(* IEC 61131-3 sources: programs/VI-54/VI-54_20171205/VI-54_20171205/Stations/PLC_VI54/VI-54_171014/Class/_DriveActValues, 1 file *)

(* ---- _DriveActValues.st ---- *)
(*!
<Class
	Name               = "_DriveActValues"
	Revision           = "1.13"
	RealtimeTask       = "false"
	CyclicTask         = "true"
	DefCyclictime      = "100 ms"
	BackgroundTask     = "false"
	Sigmatek           = "true"
	OSInterface        = "false"
	HighPriority       = "false"
	Automatic          = "false"
	UpdateMode         = "Prescan"
	IconPath           = ".\Class\_DriveMngBase\Drive.ico"
	SharedCommandTable = "true"
	Objectsize         = "(570,1920)"
	Comment            = "displays the actual values of the connected Drive">
	<Channels>
		<Server Name="I_BCC" Visualized="true" Initialize="false" WriteProtected="true" Retentive="false" Comment="Para-Nr : 182&#13;&#10;Unit  : [-]&#13;&#10;Checksum of all parameters for data integrity check&#13;&#10;"/>
		<Server Name="I_BITS" Visualized="true" Initialize="false" WriteProtected="true" Retentive="false" Comment="Para-Nr : 205&#13;&#10;Unit  : [-]&#13;&#10;BIT 0 ... PLL BIT0:&#13;&#10;BIT 1 ... PLL BIT1:&#13;&#10;00=PLL locked;&#13;&#10;01=PLL locked, more than half of the pll range is used (frequency to high);&#13;&#10;10=PLL locked, less than half of the pll range is used (frequency to low);&#13;&#10;11=PLL not locked&#13;&#10;BIT 2 ... Digital Input 6: LOCK &amp; ENABLE &amp; ENABLE_BRAKE&#13;&#10;BIT 3 ... IGBT Voltage (LOCK)&#13;&#10;BIT 4 ... ENABLE Input&#13;&#10;BIT 5 ... ENABLE_BRAKE Input&#13;&#10;BIT 6 ... Digital Input 1&#13;&#10;BIT 7 ... Digital Input 2&#13;&#10;BIT 8 ... Digital Input 3&#13;&#10;BIT 9 ... Digital Input 4&#13;&#10;BIT10 ... Digital Input 5"/>
		<Server Name="I_CAP" Visualized="true" Initialize="false" WriteProtected="true" Retentive="false" Comment="Para-Nr : 202&#13;&#10;Unit  : [-]&#13;&#10;Motorposition at the last edge of the capture input&#13;&#10;The selection of the input and the edge (rising/falling) is done by [A-CAPREF].&#13;&#10;&#13;&#10;If a capture happens, the corresponding bit in the statusword is toggled (statusword see [A-VALTT1] and [A-VALTT2]).&#13;&#10;"/>
		<Server Name="I_CAP4" Visualized="true" Initialize="false" WriteProtected="true" Retentive="false" Comment="Para-Nr : 203&#13;&#10;Unit  : [-]&#13;&#10;Motorposition at the last edge of the common capture input 4&#13;&#10;&#13;&#10;If a capture happens, the corresponding bit in the statusword is toggled (statusword see [A-VALTT1] and [A-VALTT2])."/>
		<Server Name="I_CAPENC" Visualized="true" Initialize="false" WriteProtected="true" Retentive="false" Comment="Para-Nr : 204&#13;&#10;Unit  : [-]&#13;&#10;Position of the second encoder at the last edge at the capture input&#13;&#10;The selection of the input and the edge (rising/falling) is done by A-CAPREF.&#13;&#10;&#13;&#10;If a capture happens, the corresponding bit in the statusword is toggled (statusword see A-VALTT1 and A-VALTT2)."/>
		<Server Name="I_DERROR" Visualized="true" Initialize="false" WriteProtected="true" Retentive="false" Comment="Para-Nr : 201&#13;&#10;Unit  : [-]&#13;&#10;Description : Internal Drive Errors&#13;&#13;&#10;&#13;&#13;&#10;MDD,SDD - Drives &#13;&#10;=============================================================================================&#13;&#10;Bit   0 SSI_ERROR (not supported by MDD 100)(additional Information to the Host Communication Error in [I-STATUS])&#13;&#10;Bit   1 HOST_ERROR (not supported by MDD 100)(additional Information to the Host Communication Error in [I-STATUS])&#13;&#10;Bit   2 SHORT_ERROR (short of the power stage)&#13;&#10;Bit   3 RAM_ERROR (error in the code ram area)&#13;&#10;Bit   4 FPGA_WATCHDOG_ERROR (not supported by MDD 100)(is set by the fpga watchdog mechanism)&#13;&#10;Bit   5 ADOFF_ERROR (not supported by MDD 100)(the offset of the motor current is to high)&#13;&#10;Bit   6 VCC18_ERROR (Phasing Direction Error, set when the motor turns in the wrong direction after commutation)&#13;&#10;Bit   7 VCCE_ERROR (Internal Encoder Error)&#13;&#10;Bit   8 ASMFU_IMAX_ERROR (is set if the asynchronous motor current is to high)&#13;&#10;Bit   9 PHASING_SIGNAL_STRENGTH_ERROR (Phasing Signal Strengh Error, more detailed information in Drive help parameter description I-DERROR)&#13;&#10;Bit  10 PHASING_POSITION_ERROR (is set when the position of the motor changes too drastically durin commutation)&#13;&#10;Bit  11 REGEN_ERROR (is set if the regen resistor can not be turned off)&#13;&#10;Bit  12 ENCODER_COUNTER_ERROR (not supported by MDD 100)(is set if the encoder counter check detects a fault)&#13;&#10;Bit  13 SIN_COS_COMMUT_ERROR (is set if a communication error exceeds 50ms)&#13;&#10;Bit  14 LVDS_ERROR (MDD only, is set if a communication error occurs between master and slave)&#13;&#10;Bit  15 PHASING_PHASE_SHIFT_ERROR (is set when the distance between the maximum positive/negative feedback peaks does not equal 180° +- 8°)&#13;&#10;Bit  16 PHASING_FOURIER_SIGNAL_ERROR (fourier signal cannot be calculated)&#13;&#10;&#13;&#10;DC06x&#13;&#10;=============================================================================================&#13;&#10;Bit   2 SHORT_ERROR (short of the power stage)&#13;&#10;Bit  13 FEEDBACK_ADC (feedback resolver values are not valid)(only DC061)&#13;&#10;Bit  15 SAFETY_ERROR  (safety error)&#13;&#10;Bit  16 SAFETY_WARNING (safety warning) &#13;&#10;Bit  21 Z_IMPULS_ERROR  (the z-impuls did not appeared within the time frame) (only DC062)&#13;&#10;Bit  23 FEEDBACK_SUPPLY (the feedback supply voltage fell below 15V)(only DC062)&#13;&#10;&#13;&#10;&#13;&#10;For more detailed informations, look at the parameter description of I-DERROR (201) in the Drive Help.&#13;&#13;&#10;These bits cause the Drive Error Ramp/Drive Error No Ramp in [I-STATUS]."/>
		<Server Name="I_FBB" Visualized="true" Initialize="false" WriteProtected="true" Retentive="false" Comment="Para-Nr : 208&#13;&#10;Unit  : [-]&#13;&#10;Actual value Feedback bits&#13;&#10;&#13;&#10;Bit0: Toggle status bit for the cyclic monitoring of the error status for EnDat and Hiperface encoders. See A-FB.&#13;&#10;Bit1: Status bit for the K-FBRW 5 command (Read offset from encoder). If this command was executed, Bit1 = 1. &#13;&#10;Bit2..15: Reserve&#13;&#10;Bit16..31: In these 2 bytes, the internal encoder error codes are stored as long as the K-FBRW 4 command was executed or the cyclic error status monitor is active (A-FB).&#13;&#10;"/>
		<Server Name="I_FPOS" Visualized="true" Initialize="false" WriteProtected="true" Retentive="false" Comment="Para-Nr : 177&#13;&#10;Unit  : [-]&#13;&#10;Description : Resolver angle&#13;&#10;&#13;&#10;"/>
		<Server Name="I_I2T" Visualized="true" Initialize="false" WriteProtected="true" Retentive="false" Comment="Para-Nr : 193&#13;&#10;Unit  : [%]&#13;&#10;Description : Actual value of I2T of the power stage in % of [C-ICONT]&#13;&#13;&#10;&#13;&#13;&#10;The i2t-mechanism of the drive limits the current and the continuous current is always limited to the value of [C-ICONT].&#13;&#10;"/>
		<Server Name="I_IA" Visualized="true" Initialize="false" WriteProtected="true" Retentive="false" Comment="Para-Nr : 178 &#13;&#10;Unit  : [-]&#13;&#10;AD-value Ia (only for test purpose)&#13;&#10;"/>
		<Server Name="I_IB" Visualized="true" Initialize="false" WriteProtected="true" Retentive="false" Comment="Para-Nr : 179&#13;&#10;Unit  : [-]&#13;&#10;AD-value Ib (only for test purpose)"/>
		<Server Name="I_ICMD" Visualized="true" Initialize="false" WriteProtected="true" Retentive="false" Comment="Para-Nr : 194&#13;&#10;Unit  : [mA]&#13;&#10;Description : Current set point in Q - direction"/>
		<Server Name="I_ICONT" Visualized="true" Initialize="false" WriteProtected="true" Retentive="false" Comment="Para-Nr : 186&#13;&#10;Unit  : [mA]&#13;&#10;Description : Drive continuos current&#13;&#10;"/>
		<Server Name="I_ID" Visualized="true" Initialize="false" WriteProtected="true" Retentive="false" Comment="Para-Nr : 192&#13;&#10;Unit  : [mA]&#13;&#10;Description : Actual value of the current in D - direction&#13;&#10;"/>
		<Server Name="I_INT1" Visualized="true" Initialize="false" WriteProtected="true" Retentive="false" Comment="Para-Nr : 206&#13;&#10;Unit  : [-]&#13;&#10;Internal Actual Value 1&#13;&#10;&#13;&#10;A-INT1 defines which internal actual value is displayed here.&#13;&#10;&#13;&#10;See also I-INT2."/>
		<Server Name="I_INT2" Visualized="true" Initialize="false" WriteProtected="true" Retentive="false" Comment="Para-Nr : 207&#13;&#10;Unit  : [-]&#13;&#10;Internal Actual Value 2&#13;&#10;&#13;&#10;A-INT2 defines which internal actual value is displayed here.&#13;&#10;&#13;&#10;See also I-INT1."/>
		<Server Name="I_IPEAK" Visualized="true" Initialize="false" WriteProtected="true" Retentive="false" Comment="Para-Nr : 185&#13;&#10;Unit  : [mA]&#13;&#10;Description : Drive peak current&#13;&#10;"/>
		<Server Name="I_IQ" Visualized="true" Initialize="false" WriteProtected="true" Retentive="false" Comment="Para-Nr : 191&#13;&#10;Unit  : [mA]&#13;&#10;Description : Actual value of the current in Q - direction&#13;&#10;"/>
		<Server Name="I_MPOS" Visualized="true" Initialize="false" WriteProtected="true" Retentive="false" Comment="Para-Nr : 180&#13;&#10;Unit  : [-]&#13;&#10;Description : Actual multiturn position  in 1/8 of a revolution (available only with [M-TYPE] = 1)"/>
		<Server Name="I_N" Visualized="true" Initialize="false" WriteProtected="true" Retentive="false" Comment="Para-Nr : 197&#13;&#10;Unit  : [rpm]&#13;&#10;Description : Actual speed unsmoothed&#13;&#10;"/>
		<Server Name="I_NCMD" Visualized="true" Initialize="false" WriteProtected="true" Retentive="false" Comment="Para-Nr : 190&#13;&#10;Unit  : [rpm]&#13;&#10;Description : Speed set point&#13;&#10;"/>
		<Server Name="I_NFILT" Visualized="true" Initialize="false" WriteProtected="true" Retentive="false" Comment="Para-Nr : 198&#13;&#10;Unit  : [rpm]&#13;&#10;Description : Actual speed smoothed by [V-T]&#13;&#10;"/>
		<Server Name="I_PBAL" Visualized="true" Initialize="false" WriteProtected="true" Retentive="false" Comment="Para-Nr : 196&#13;&#10;Unit  : [W]&#13;&#10;Description : Actual regen power&#13;&#13;&#10;This value is influenced by [G-RBAL].&#13;&#10;"/>
		<Server Name="I_PCMD" Visualized="true" Initialize="false" WriteProtected="true" Retentive="false" Comment="Para-Nr : 174&#13;&#10;Unit  : [-]&#13;&#10;Description : Position setpoint&#13;&#10;"/>
		<Server Name="I_PE" Visualized="true" Initialize="false" WriteProtected="true" Retentive="false" Comment="Para-Nr : 175&#13;&#10;Unit  : [-]&#13;&#10;Description : Position error&#13;&#10;&#13;&#10;"/>
		<Server Name="I_POS" Visualized="true" Initialize="false" WriteProtected="true" Retentive="false" Comment="Para-Nr : 176&#13;&#10;Unit  : [-]&#13;&#10;Description : Actual position (internal 64 bit position scaled by [P-PSCALE])&#13;&#10;&#13;&#10;"/>
		<Server Name="I_STATUS" Visualized="true" Initialize="false" WriteProtected="true" Retentive="false" Comment="Para-Nr : 199&#13;&#10;Unit  : [-]&#13;&#10;Description : Status register:&#13;&#13;&#10;&#13;&#13;&#10;Bit  0   Mains phase (1-phase supply)&#13;&#10;Bit  1   Mains fault&#13;&#10;Bit  2   Motor axis over-current&#13;&#10;Bit  3   Over voltage DC-Link&#13;&#10;Bit  4   Under voltage DC-link&#13;&#10;Bit  5   Motor axis phase failure&#13;&#10;Bit  6   Holding brake error&#13;&#10;Bit  7   Holding brake switch damaged&#13;&#10;Bit  8   reserved&#13;&#10;Bit  9   Motor thermostat&#13;&#10;Bit 10  Ambient temperature&#13;&#10;Bit 11  Heat sink temperature&#13;&#10;Bit 12  Feedback Error&#13;&#10;Bit 13  Commutation error&#13;&#10;Bit 14  Over speed&#13;&#10;Bit 15  Contouring Error&#13;&#10;Bit 16  Trajectory Error&#13;&#10;Bit 17  Host Communication Error&#13;&#10;Bit 18  Drive Error Ramp, for additional information see [I-DERROR]&#13;&#10;Bit 19  Drive Error No Ramp, for additional information see [I-DERROR]&#13;&#10;Bit 20  External Enable Locked Error&#13;&#10;Bit 21  IGBT Driver Voltage Error&#13;&#10;Bit 22  max. Regen Power Error&#13;&#10;Bit 23  24V Brake Supply Error&#13;&#10;Bit 24  reserved&#13;&#10;Bit 25  I2T-Error&#13;&#10;Bit 26  Motor Temperature Warning&#13;&#10;Bit 27  Motor Parameter Error&#13;&#10;Bit 28  Multi-Turn Position Error&#13;&#10;Bit 29  Max Sum Power Limitation&#13;&#10;Bit 30  Speed Controler in Saturation&#13;&#10;Bit 31  Fan Error &#13;&#10;&#13;&#13;&#10;The masks  [G-MASKE1], [G-MASKE2], [G-MASKW] and [G-MASKD] &#13;&#10;define if the corresponding bit of I-STATUS causes a cast of the motor, a ramp stop of the motor, a warning or nothing.&#13;&#13;&#10;This errors can be cleared with [K-CLRF].&#13;&#10;For more detailed informations, look at the parameter description of I-STATUS(199) in the Drive Help.&#13;&#10;"/>
		<Server Name="I_TEMPE" Visualized="true" Initialize="false" WriteProtected="true" Retentive="false" Comment="Para-Nr : 184&#13;&#10;Unit  : [°C]&#13;&#10;Description : Actual ambient temperature&#13;&#10;"/>
		<Server Name="I_TEMPK" Visualized="true" Initialize="false" WriteProtected="true" Retentive="false" Comment="Para-Nr : 183&#13;&#10;Unit  : [°C]&#13;&#10;Description : Actual heat sink temperature&#13;&#10;&#13;&#10;"/>
		<Server Name="I_TEMPM" Visualized="true" Initialize="false" WriteProtected="true" Retentive="false" Comment="Para-Nr : 181&#13;&#10;Unit  : [Ohm]&#13;&#10;Description : Actual value of the PTC in the motor winding &#13;&#10;"/>
		<Server Name="I_VBUS" Visualized="true" Initialize="false" WriteProtected="true" Retentive="false" Comment="Para-Nr : 195&#13;&#10;Unit  : [V]&#13;&#10;Description : Actual DC-link voltage&#13;&#10;"/>
	</Channels>
	<RevDoku>
		<Owner Company="Sigmatek" Author="HasHan"/>
		<Dokumentation Revision="1.13" Date="08.11.2016" Author="ZoePat" Company="Sigmatek" Description="Client &quot;DriveAxis&quot; is now not required."/>
		<Dokumentation Revision="1.12" Date="16.06.2015" Author="EisMic" Company="Sigmatek" Description="Updated description from I-STATUSand I-DERROR Bits."/>
		<Dokumentation Revision="1.11" Date="06.10.2014" Author="LanSte" Company="Sigmatek" Description="Added support for drive parameters P208 amd P122"/>
		<Dokumentation Revision="1.10" Date="04.12.2013" Author="ObeChr" Company="Sigmatek" Description="Added missing Bits in Type for Server I-STATUS + I-DERROR"/>
		<Dokumentation Revision="1.0" Date="05.08.2009" Author="HasHan" Company="Sigmatek" Description="Creation"/>
	</RevDoku>
	<Network Name="_DriveActValues">
		<!-- List of Components in this network -->
		<Components>
			<Object
				Name       = "_base"
				Class      = "_DriveParaBase"
				Position   = "(218,120)"
				Visualized = "false">
				<Channels>
					<Server Name="State"/>
					<Client Name="DriveAxis"/>
					<Client Name="ErrorCode"/>
				</Channels>
			</Object>
		</Components>
		<Comments>
		</Comments>
		<!-- List of Connections in this network -->
		<Connections>
			<Connection Source="this.State" Destination="_base.State" Vertices="(740,210),(568,210),"/>
			<Connection Source="_base.DriveAxis" Destination="this.DriveAxis" Vertices="(218,210),(38,210),"/>
			<Connection Source="_base.ErrorCode" Destination="this.ErrorCode" Vertices="(218,270),(38,270),"/>
		</Connections>
		<!-- Headerfiles -->
		<Options>
		</Options>
	</Network>
</Class>
*)
#pragma using _DriveParaBase

_DriveActValues : CLASS
: _DriveParaBase
  //Servers:
	I_PCMD 	: SvrCh_DINT;
	I_PE 	: SvrCh_DINT;
	I_POS 	: SvrCh_DINT;
	I_FPOS 	: SvrCh_DINT;
	I_MPOS 	: SvrCh_DINT;
	I_TEMPM 	: SvrCh_DINT;
	I_TEMPK 	: SvrCh_DINT;
	I_TEMPE 	: SvrCh_DINT;
	I_IPEAK 	: SvrCh_DINT;
	I_ICONT 	: SvrCh_DINT;
	I_NCMD 	: SvrCh_DINT;
	I_IQ 	: SvrCh_DINT;
	I_ID 	: SvrCh_DINT;
	I_I2T 	: SvrCh_DINT;
	I_ICMD 	: SvrCh_DINT;
	I_VBUS 	: SvrCh_DINT;
	I_PBAL 	: SvrCh_DINT;
	I_N 	: SvrCh_DINT;
	I_NFILT 	: SvrCh_DINT;
	I_STATUS 	: SvrCh__SDDISTATE;
	I_DERROR 	: SvrCh__SDDIDERROR;
	I_BCC 	: SvrCh_DINT;
	I_IA 	: SvrCh_DINT;
	I_IB 	: SvrCh_DINT;
	I_CAP 	: SvrCh_DINT;
	I_CAP4 	: SvrCh_DINT;
	I_CAPENC 	: SvrCh_DINT;
	I_BITS 	: SvrCh_DINT;
	I_INT1 	: SvrCh_DINT;
	I_INT2 	: SvrCh_DINT;
	I_FBB 	: SvrCh_DINT;
  //Clients:
  //Variables:
		TimeMarkFast 	: UDINT;
		ActValSSW 	: DINT;
		bdActValActive : BDINT
		[
		  1 bI_PCMD,
		  2 bI_PE,
		  3 bI_POS,
		  4 bI_FPOS,
		  5 bI_MPOS,
		  6 bI_TEMPM,
		  7 bI_TEMPK,
		  8 bI_TEMPE,
		  9 bI_IPEAK,
		  10 bI_ICONT,
		  11 bI_NCMD,
		  12 bI_IQ,
		  13 bI_ID,
		  14 bI_I2T,
		  15 bI_ICMD,
		  16 bI_VBUS,
		  17 bI_PBAL,
		  18 bI_N,
		  19 bI_NFILT,
		  20 I_STATUS,
		  21 bI_I_DERROR,
		];

  //Functions:

	FUNCTION VIRTUAL GLOBAL Init;

	FUNCTION VIRTUAL GLOBAL CyWork
		VAR_INPUT
			EAX 	: UDINT;
		END_VAR
		VAR_OUTPUT
			state (EAX) 	: UDINT;
		END_VAR;

	FUNCTION VIRTUAL GLOBAL RefreshPara
		VAR_INPUT
			usParaNr 	: USINT;
			dValue 	: DINT;
		END_VAR;

	FUNCTION GLOBAL ActValProc;
  //Tables:
	FUNCTION @STD
		VAR_OUTPUT
			ret_code	: CONFSTATES;
		END_VAR;
	FUNCTION GLOBAL TAB @CT_;
END_CLASS;

FUNCTION VIRTUAL GLOBAL _DriveActValues::CyWork
	VAR_INPUT
		EAX 	: UDINT;
	END_VAR
	VAR_OUTPUT
		state (EAX) 	: UDINT;
	END_VAR

	state:= READY;

  if (IsAxisConnected() = TRUE) & (DriveAxis.AxOkay() = true) & (DriveAxis.IsOnline() = true) then
    ActValProc();
    if DriveAxis <> READY then
      DriveAxis := READY;
    end_if;
  else
    this^.State  := ERROR;
    DriveAxis    := ERROR;
    ActValSSW    := SDD_I_PCMD;
    AnzASyncPara := 0;
  end_if;

END_FUNCTION

FUNCTION GLOBAL _DriveActValues::ActValProc

  if ops.tabsolute - TimeMarkFast >= ACTVALTIMEFAST then

    TimeMarkFast := ops.tabsolute;
    case ActValSSW of
    SDD_I_PCMD :
      SetASyncCmd(ParaNr:= SDD_I_PCMD, ParaRdWr:= 0, ParaValue:= 0, pThis:= this);
      ActValSSW := SDD_I_PE;

    SDD_I_PE :
      SetASyncCmd(ParaNr:= SDD_I_PE, ParaRdWr:= 0, ParaValue:= 0, pThis:= this);
      ActValSSW := SDD_I_POS;

    SDD_I_POS :
      SetASyncCmd(ParaNr:= SDD_I_POS, ParaRdWr:= 0, ParaValue:= 0, pThis:= this);
      ActValSSW := SDD_I_FPOS;

    SDD_I_FPOS :
      SetASyncCmd(ParaNr:= SDD_I_FPOS, ParaRdWr:= 0, ParaValue:= 0, pThis:= this);
      ActValSSW := SDD_I_MPOS;

    SDD_I_MPOS :
      SetASyncCmd(ParaNr:= SDD_I_MPOS, ParaRdWr:= 0, ParaValue:= 0, pThis:= this);
      ActValSSW := SDD_I_TEMPM;

    SDD_I_TEMPM :
      SetASyncCmd(ParaNr:= SDD_I_TEMPM, ParaRdWr:= 0, ParaValue:= 0, pThis:= this);
      ActValSSW := SDD_I_TEMPK;

    SDD_I_TEMPK :
      SetASyncCmd(ParaNr:= SDD_I_TEMPK, ParaRdWr:= 0, ParaValue:= 0, pThis:= this);
      ActValSSW := SDD_I_TEMPE;

    SDD_I_TEMPE :
      SetASyncCmd(ParaNr:= SDD_I_TEMPE, ParaRdWr:= 0, ParaValue:= 0, pThis:= this);
      ActValSSW := SDD_I_IPEAK;

    SDD_I_IPEAK :
      SetASyncCmd(ParaNr:= SDD_I_IPEAK, ParaRdWr:= 0, ParaValue:= 0, pThis:= this);
      ActValSSW := SDD_I_ICONT;

    SDD_I_ICONT :
      SetASyncCmd(ParaNr:= SDD_I_ICONT, ParaRdWr:= 0, ParaValue:= 0, pThis:= this);
      ActValSSW := SDD_I_NCMD;

    SDD_I_NCMD :
      SetASyncCmd(ParaNr:= SDD_I_NCMD, ParaRdWr:= 0, ParaValue:= 0, pThis:= this);
      ActValSSW := SDD_I_IQ;

    SDD_I_IQ :
      SetASyncCmd(ParaNr:= SDD_I_IQ, ParaRdWr:= 0, ParaValue:= 0, pThis:= this);
      ActValSSW := SDD_I_ID;

    SDD_I_ID :
      SetASyncCmd(ParaNr:= SDD_I_ID, ParaRdWr:= 0, ParaValue:= 0, pThis:= this);
      ActValSSW := SDD_I_I2T;

    SDD_I_I2T :
      SetASyncCmd(ParaNr:= SDD_I_I2T, ParaRdWr:= 0, ParaValue:= 0, pThis:= this);
      ActValSSW := SDD_I_ICMD;

    SDD_I_ICMD :
      SetASyncCmd(ParaNr:= SDD_I_ICMD, ParaRdWr:= 0, ParaValue:= 0, pThis:= this);
      ActValSSW := SDD_I_VBUS;

    SDD_I_VBUS :
      SetASyncCmd(ParaNr:= SDD_I_VBUS, ParaRdWr:= 0, ParaValue:= 0, pThis:= this);
      ActValSSW := SDD_I_PBAL;

    SDD_I_PBAL :
      SetASyncCmd(ParaNr:= SDD_I_PBAL, ParaRdWr:= 0, ParaValue:= 0, pThis:= this);
      ActValSSW := SDD_I_N;

    SDD_I_N :
      SetASyncCmd(ParaNr:= SDD_I_N, ParaRdWr:= 0, ParaValue:= 0, pThis:= this);
      ActValSSW := SDD_I_NFILT;

    SDD_I_NFILT :
      SetASyncCmd(ParaNr:= SDD_I_NFILT, ParaRdWr:= 0, ParaValue:= 0, pThis:= this);
      ActValSSW := SDD_I_STATUS;

    SDD_I_STATUS :
      SetASyncCmd(ParaNr:= SDD_I_STATUS, ParaRdWr:= 0, ParaValue:= 0, pThis:= this);
      ActValSSW := SDD_I_DERROR;

    SDD_I_DERROR :
      SetASyncCmd(ParaNr:= SDD_I_DERROR, ParaRdWr:= 0, ParaValue:= 0, pThis:= this);
      ActValSSW := SDD_I_CAP;

    SDD_I_CAP :
      SetASyncCmd(ParaNr:= SDD_I_CAP, ParaRdWr:= 0, ParaValue:= 0, pThis:= this);
      ActValSSW := SDD_I_CAP4;

    SDD_I_CAP4 :
      SetASyncCmd(ParaNr:= SDD_I_CAP4, ParaRdWr:= 0, ParaValue:= 0, pThis:= this);
      ActValSSW := SDD_I_CAPENC;

    SDD_I_CAPENC :
      SetASyncCmd(ParaNr:= SDD_I_CAPENC, ParaRdWr:= 0, ParaValue:= 0, pThis:= this);
      ActValSSW := SDD_I_BITS;

    SDD_I_BITS :
      SetASyncCmd(ParaNr:= SDD_I_BITS, ParaRdWr:= 0, ParaValue:= 0, pThis:= this);
      ActValSSW := SDD_I_INT1;

    SDD_I_INT1 :
      SetASyncCmd(ParaNr:= SDD_I_INT1, ParaRdWr:= 0, ParaValue:= 0, pThis:= this);
      ActValSSW := SDD_I_INT2;

    SDD_I_INT2 :
      SetASyncCmd(ParaNr:= SDD_I_INT2, ParaRdWr:= 0, ParaValue:= 0, pThis:= this);
      ActValSSW := SDD_I_IA;

    SDD_I_IA :
      SetASyncCmd(ParaNr:= SDD_I_IA, ParaRdWr:= 0, ParaValue:= 0, pThis:= this);
      ActValSSW := SDD_I_IB;

    SDD_I_IB :
      SetASyncCmd(ParaNr:= SDD_I_IB, ParaRdWr:= 0, ParaValue:= 0, pThis:= this);
      ActValSSW := SDD_I_BCC;

    SDD_I_BCC :
      SetASyncCmd(ParaNr:= SDD_I_BCC, ParaRdWr:= 0, ParaValue:= 0, pThis:= this);
      ActValSSW := SDD_I_FBB;

    SDD_I_FBB :
      SetASyncCmd(ParaNr:= SDD_I_FBB, ParaRdWr:= 0, ParaValue:= 0, pThis:= this);
      ActValSSW := SDD_I_PCMD;

    end_case;
  end_if;

END_FUNCTION

FUNCTION VIRTUAL GLOBAL _DriveActValues::RefreshPara
	VAR_INPUT
		usParaNr 	: USINT;
		dValue 	: DINT;
	END_VAR

  case usParaNr of

  SDD_I_PCMD :
    I_PCMD := dValue;

  SDD_I_PE :
    I_PE := dValue;

  SDD_I_POS :
    I_POS := dValue;

  SDD_I_FPOS :
    I_FPOS := dValue;

  SDD_I_MPOS :
    I_MPOS := dValue;

  SDD_I_TEMPM :
    I_TEMPM := dValue;

  SDD_I_TEMPK :
    I_TEMPK := dValue;

  SDD_I_TEMPE :
    I_TEMPE := dValue;

  SDD_I_IPEAK :
    I_IPEAK := dValue;

  SDD_I_ICONT :
    I_ICONT := dValue;

  SDD_I_NCMD :
    I_NCMD := dValue;

  SDD_I_IQ :
    I_IQ := dValue;

  SDD_I_ID :
    I_ID := dValue;

  SDD_I_I2T :
    I_I2T := dValue;

  SDD_I_ICMD :
    I_ICMD := dValue;

  SDD_I_VBUS :
    I_VBUS := dValue;

  SDD_I_PBAL :
    I_PBAL := dValue;

  SDD_I_N :
    I_N := dValue;

  SDD_I_NFILT :
    I_NFILT := dValue;

  SDD_I_STATUS :
    I_STATUS$DINT := dValue;

  SDD_I_DERROR :
    I_DERROR$DINT := dValue;

  SDD_I_CAP :
    I_CAP := dValue;

  SDD_I_CAP4 :
    I_CAP4 := dValue;

  SDD_I_CAPENC :
    I_CAPENC := dValue;

  SDD_I_BITS :
    I_BITS := dValue;

  SDD_I_INT1 :
    I_INT1 := dValue;

  SDD_I_INT2 :
    I_INT2 := dValue;

  SDD_I_IA :
    I_IA := dValue;

  SDD_I_IB :
    I_IB := dValue;

  SDD_I_BCC :
    I_BCC := dValue;

  SDD_I_FBB :
    I_FBB := dValue;

  end_case;

END_FUNCTION

FUNCTION VIRTUAL GLOBAL _DriveActValues::Init

  // call base method
  _DriveParaBase::Init();

  if _firstscan then
    ActValSSW := SDD_I_PCMD;
  end_if;

END_FUNCTION
